Omron CX-Programmer project NewProject (CX-Programmer 9.50)

# PLC SMT: CQM1H CPU11

## Global symbols (name address type ; comment)
0.00 BOOL  ; Sensor start
0.01 BOOL  ; sensor 1
0.02 BOOL  ; sensor 2
0.03 BOOL  ; sensor3
0.04 BOOL  ; sensor akhir
100.00 BOOL  ; Conveyor ON
100.01 BOOL  ; enable mikro kanan
100.02 BOOL  ; enable mikro kiri
200.01 BOOL  ; temp kanan
200.02 BOOL  ; temp kiri
200.03 BOOL  ; prepare stepper
200.04 BOOL  ; enable stepper
200.05 BOOL  ; gerak kanan
200.06 BOOL  ; gerak kiri

## Program NewProgram1 (no task)

### Section Section1

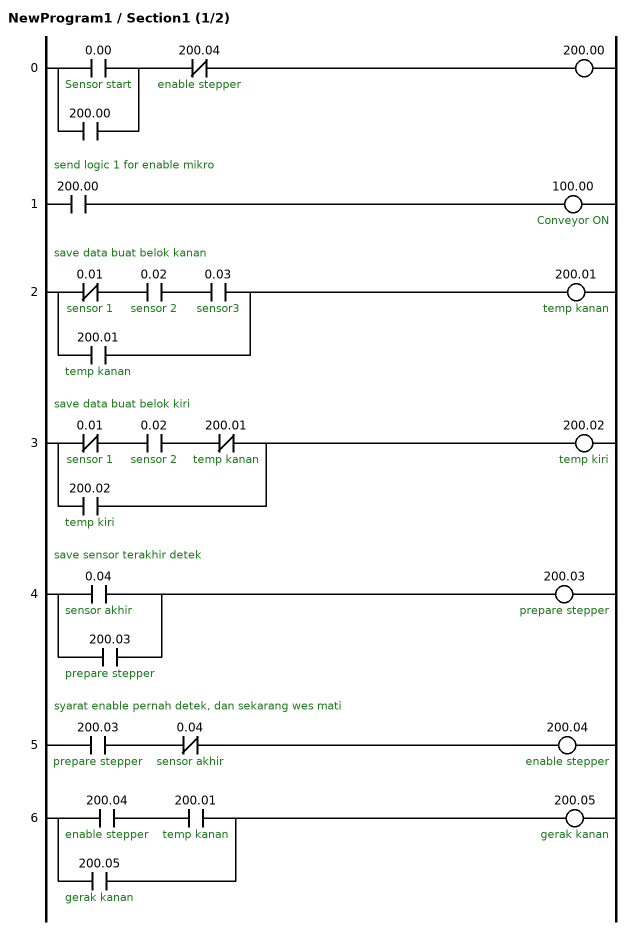
; rung 0
LD 0.00  ; Sensor start
OR 200.00
ANDNOT 200.04  ; enable stepper
OUT 200.00
; rung 1: send logic 1 for enable mikro
LD 200.00
OUT 100.00  ; Conveyor ON
; rung 2: save data buat belok kanan
LDNOT 0.01  ; sensor 1
AND 0.02  ; sensor 2
AND 0.03  ; sensor3
OR 200.01  ; temp kanan
OUT 200.01  ; temp kanan
; rung 3: save data buat belok kiri
LDNOT 0.01  ; sensor 1
AND 0.02  ; sensor 2
ANDNOT 200.01  ; temp kanan
OR 200.02  ; temp kiri
OUT 200.02  ; temp kiri
; rung 4: save sensor terakhir detek
LD 0.04  ; sensor akhir
OR 200.03  ; prepare stepper
OUT 200.03  ; prepare stepper
; rung 5: syarat enable pernah detek, dan sekarang wes mati
LD 200.03  ; prepare stepper
ANDNOT 0.04  ; sensor akhir
OUT 200.04  ; enable stepper
; rung 6
LD 200.04  ; enable stepper
AND 200.01  ; temp kanan
OR 200.05  ; gerak kanan
OUT 200.05  ; gerak kanan

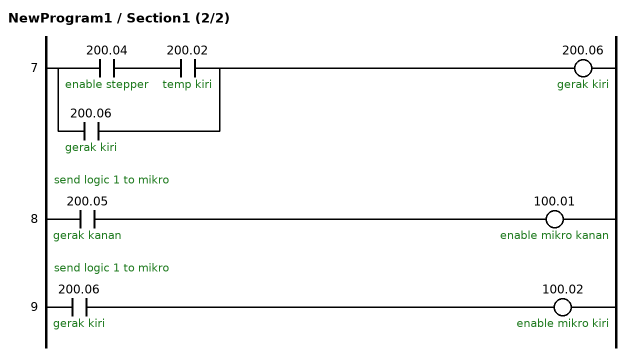
; rung 7
LD 200.04  ; enable stepper
AND 200.02  ; temp kiri
OR 200.06  ; gerak kiri
OUT 200.06  ; gerak kiri
; rung 8: send logic 1 to mikro
LD 200.05  ; gerak kanan
OUT 100.01  ; enable mikro kanan
; rung 9: send logic 1 to mikro
LD 200.06  ; gerak kiri
OUT 100.02  ; enable mikro kiri

### Section END
; rung 0
END(01)